FUNCTION getUsint : BOOL
VAR_INPUT
END_VAR
VAR
END_VAR
VAR_IN_OUT
	usintRef : USINT;
	bufferRef : UDINT;
END_VAR

	memcpy(ADR(usintRef), bufferRef, SIZEOF(USINT));
	bufferRef := bufferRef + SIZEOF(USINT);
	getUsint := TRUE;

END_FUNCTION

(* stored: Version 1.1.0.1, ProductVersion 3.1.4024.3
   POU getUsint: Id {2dcf5877-62b1-0fdb-3782-feefb6918a0b}, SpecialFunc None *)
